// TIA Portal V20 export
TYPE "LPFE_typeWarning"
// stored: Access Published, Namespace PFE
   STRUCT
      Maintenance : Struct
         MW : Struct
            "kDiag.Alarm.MaintWarnPLCSW" : Int := 201;   // PLC Software Maintenance Warning (Minor Fault ...)
            "kDiag.Alarm.MaintWarnPLCHW" : Int := 202;   // PLC Hardware Maintenance Warning (Battery Low ...)
            "kDiag.Alarm.MaintWarnGeneral" : Int := 204;   // Maintenance Warning General
         END_STRUCT;
      END_STRUCT;
      Production : Struct
         PW : Struct
            "kDiag.Alarm.ProdWarn" : Int := 205;   // Production Warning
            "kDiag.Alarm.ProdWarnAndon" : Int := 206;
         END_STRUCT;
      END_STRUCT;
      Tooling : Struct
         LW : Struct
            "kDiag.Alarm.ToolWarn" : Int := 210;   // Tooling Warning
         END_STRUCT;
      END_STRUCT;
      Quality : Struct
         QW : Struct
            "kDiag.Alarm.QualWarn" : Int := 215;   // Quality Warning
            "kDiag.Alarm.QualWarnAndon" : Int := 216;
         END_STRUCT;
      END_STRUCT;
      Throughput : Struct
         TW : Struct
            "kDiag.Alarm.TputWarn" : Int := 220;   // Thruput Warning
         END_STRUCT;
      END_STRUCT;
      System : Struct
         SW : Struct
            "kDiag.Alarm.SysWarn" : Int := 225;   // System Warning
         END_STRUCT;
      END_STRUCT;
      Material : Struct
         AW : Struct
            "kDiag.Alarm.MatlWarn" : Int := 230;   // Material Warning
         END_STRUCT;
      END_STRUCT;
   END_STRUCT;
END_TYPE
